Fanuc KAREL source: ko00060.KL

-- PROVISIONAL review KL for V1013-1; original PC SHA256 c04fdb20e14f68945ad1fbc198353c727922b8c50ebf834bfcd0db8c96b78c07
-- Incomplete behavior may be omitted. Consult companion uncertainty JSON. Do not deploy.
PROGRAM KO00060
%NOLOCKGROUP
BEGIN
  -- UNRESOLVED_PC offsets 5-12; opcodes 9D,23
  -- UNRESOLVED_PC offsets 17-69; opcodes 27,27,49,7E,AD,27,49,7E,AD,22,31,7E,4A
  -- UNRESOLVED_PC offsets 74-78; opcodes 7F
END KO00060
